INTERFACE ITF_EM_Transport_BottomSeal_Labeller

END_INTERFACE

(* stored: Version 1.1.0.1, ProductVersion 3.1.4024.12
   Itf ITF_EM_Transport_BottomSeal_Labeller: Id {088d762d-0def-4c2e-946f-ca0e442b9987} *)
